Fanuc KAREL source: ks00041.KL

-- PROVISIONAL review KL for V1013-1; original PC SHA256 acbf64e6611860c6e68637bdfa3f79faab102675d06a6b9ae11f2cb918414bca
-- Incomplete behavior may be omitted. Consult companion uncertainty JSON. Do not deploy.
PROGRAM KS00041
%NOLOCKGROUP
BEGIN
  -- UNRESOLVED_PC offsets 5-13; opcodes 3F,75
  -- UNRESOLVED_PC offsets 18-27; opcodes 3F,75
  -- UNRESOLVED_PC offsets 32-70; opcodes 27,22,22,2A,22,2A,22,22,AF
  -- UNRESOLVED_PC offsets 75-79; opcodes 7F
END KS00041
